Universal Robots PolyScope program: group1_devs4.urp

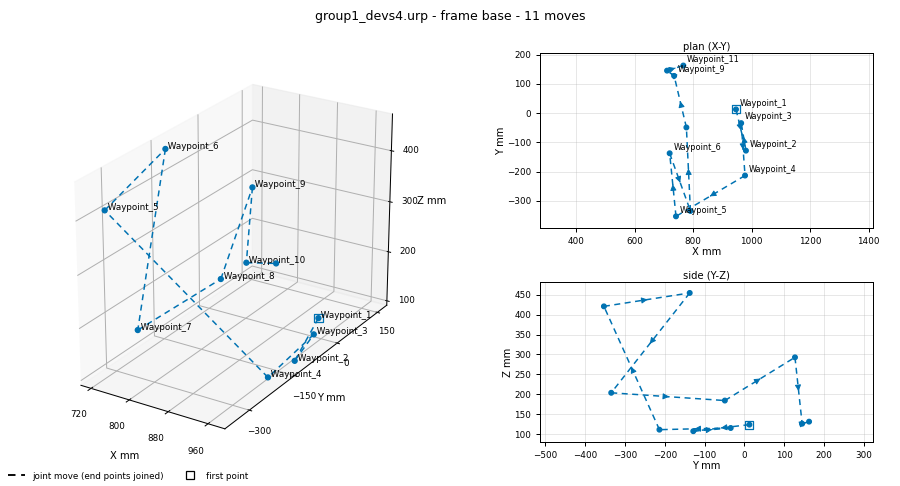
[picture p0: tool path of group1_devs4.urp in frame base, 11 of 11 moves have a stored position in this frame; points joined in program order, loops and branches not executed]
Program group1_devs4 (installation=default directory=/programs/usbdisk/Devs 4 createdIn=5.13.0 lastSavedIn=5.13.0 robotSerialNumber=20225201339)
Calibrated DH parameters: a=[-0.000118, -0.339742, -0.555336, 0.000027, 0.000053, 0]; d=[0.180691, -465.540026, 499.223902, -33.510242, 0.119749, 0.115686]; alpha=[1.571428, -0.001093, 0.003977, 1.569316, -1.571413, 0]; deltaTheta=[0, 0.982125, 5.537749, -0.236695, 0, 0]
InitVariablesNode
Robot Program (runOnlyOnce=false)
  robotState := read_port_register(200)
  If robotState≟1 (checkContinuously=true)
    ''
    MoveJ speed 60 deg/s, acceleration 80 deg/s^2 (useActiveTCP=true) feature=Base
      Waypoint Waypoint_1: motionParameters(nextMotionTime=0.5); TCP in base x=946.713 y=12.491 z=123.679 mm, rx=-0.4639 ry=-1.1141 rz=1.6522 rad; joints [1.921, -121.049, -119.24, 27.618, 114.337, -0.335] deg; TCP offset x=-0.188 y=3.576 z=256.261 mm, rx=-0.0017 ry=3.1416 rz=0 rad
      Waypoint Waypoint_2: motionParameters(nextMotionTime=0.5); TCP in base x=980.71 y=-128.525 z=107.229 mm, rx=-0.7529 ry=-0.8191 rz=1.4782 rad; joints [1.921, -121.052, -119.134, 27.615, 91.715, -0.337] deg
      Waypoint Waypoint_3: motionParameters(nextMotionTime=0.5); TCP in base x=964.479 y=-34.487 z=115.304 mm, rx=-0.5695 ry=-1.0135 rz=1.5958 rad; joints [1.93, -121.047, -119.136, 27.614, 106.484, -0.338] deg
      Waypoint Waypoint_4: motionParameters(nextMotionTime=0.5); TCP in base x=977.618 y=-213.602 z=111.091 mm, rx=-0.9027 ry=-0.6435 rz=1.3622 rad; joints [1.917, -121.05, -119.147, 27.614, 78.568, -0.337] deg
      Wait Sleep waitTime=3
  ElseIf robotState≟2 (checkContinuously=true)
    ''
    MoveJ speed 60 deg/s, acceleration 80 deg/s^2 (useActiveTCP=true) feature=Base
      Waypoint Waypoint_5: TCP in base x=741.69 y=-353.026 z=420.857 mm, rx=-0.9418 ry=-0.8359 rz=1.2032 rad; joints [-16.362, -86.436, -129.31, 12.782, 96.715, -0.51] deg
      Waypoint Waypoint_6: TCP in base x=719.998 y=-137.506 z=454.56 mm, rx=-0.5819 ry=-1.3051 rz=1.5099 rad; joints [-16.291, -86.44, -129.312, 12.765, 130.859, -0.51] deg
      Waypoint Waypoint_7: TCP in base x=791.043 y=-334.658 z=203.735 mm, rx=-1.0199 ry=-0.5304 rz=1.7725 rad; joints [-13.856, -103.486, -130.918, 20.789, 96.074, -32.515] deg
      Waypoint Waypoint_8: TCP in base x=777.24 y=-49.255 z=184.214 mm, rx=-0.7182 ry=-1.0108 rz=2.0807 rad; joints [-3.909, -103.513, -134.07, 19.639, 118.688, -32.243] deg
      Waypoint Waypoint_9: TCP in base x=735.383 y=126.93 z=292.799 mm, rx=-0.7291 ry=-1.3455 rz=1.7618 rad; joints [15.173, -99, -142.634, 45.205, 106.038, -3.575] deg
      Waypoint Waypoint_10: motionParameters(nextMotionTime=0.5); TCP in base x=711.171 y=144.944 z=126.085 mm, rx=-0.5191 ry=-1.1477 rz=1.8632 rad; joints [17.085, -109.3, -145.165, 43.91, 105.965, -3.576] deg
      Waypoint Waypoint_11: motionParameters(nextMotionTime=0.1); TCP in base x=766.803 y=162.359 z=131.214 mm, rx=-0.5473 ry=-1.1798 rz=1.8541 rad; joints [17.107, -112.93, -139.509, 43.958, 105.951, -3.592] deg
      Wait Sleep waitTime=3
